// TwinCAT 3 PLC project Units
// ProgramVersion: 3.1.4023.0
// libraries:
//   tc-tools, * (hganchev)
//   Tc2_Standard, * (Beckhoff Automation GmbH)
//   Tc2_System, * (Beckhoff Automation GmbH)
//   Tc3_Module, * (Beckhoff Automation GmbH)
//   TcUnit, * (www.tcunit.org)
// project tree:
//   / PlcTask.TcTTO
//   POUs/ UnitTests.TcPOU
//   Units/ FB_TestRange.TcPOU, FB_TestRound.TcPOU, FB_TestSplit.TcPOU
// real-time tasks:
//   TASK PlcTask: cycle T#10ms, priority 20, ADS port 350

CONFIGURATION Units
    RESOURCE PLC ON TwinCAT3
        TASK PlcTask(INTERVAL := T#10ms, PRIORITY := 20);
        PROGRAM UnitTests WITH PlcTask : UnitTests;
    END_RESOURCE
END_CONFIGURATION

// ---- POUs/UnitTests.TcPOU
PROGRAM UnitTests
VAR
	fbTestRound		: Fb_TestRound;
	fbTestSplit		: FB_TestSplit;
	fbTestRange		: FB_TestRange;
END_VAR

TcUnit.RUN();

END_PROGRAM

// ---- Units/FB_TestRound.TcPOU
FUNCTION_BLOCK FB_TestRound EXTENDS TcUnit.FB_TestSuite

//REAL
testRoundRealFail();
testRoundRealSuccess();
testRoundRealToHigh();
testRoundRealToHigh2();

// LREAL
testRoundLREALFail();
testRoundLREALSuccess();
testRoundLREALToHigh();
testRoundLREALToHigh2();

METHOD testRoundLREALFail
VAR
	rValue 		: LREAL := 1000.222222;
	Actual		: LREAL;
	Expected  	: LREAL;
END_VAR
TEST('testRoundLREALFail');

// Act
Actual := 1000.222; 

// Arrange
Expected := 1000.22;

// Assert
AssertFalse( Condition := Expected = Actual, 
			 Message := 'testRoundLREALFail Failed to round LREAL');
			 
			 
			 
TEST_FINISHED();
END_METHOD

METHOD testRoundLREALSuccess
VAR
	rValue 		: LREAL := 1000.222222;
	Actual		: LREAL;
	Expected  	: LREAL;
END_VAR
TEST('testRoundLREALSuccess');

// Act
Actual := F_ROUND_LREAL(rValue, 2); 

// Arrange
Expected := 1000.22;

// Assert
AssertEquals(Expected := Expected, 
			 Actual := Actual,
			 Message := 'testRoundLREALSuccess Failed to round LREAL');
			 
			 
			 
TEST_FINISHED();
END_METHOD

METHOD testRoundLREALToHigh
VAR
	rValue 		: LREAL := 1000.226666;
	Actual		: LREAL;
	Expected  	: LREAL;
END_VAR
TEST('testRoundLREALToHigh');

// Act
Actual := F_ROUND_LREAL(rValue, 2); 

// Arrange
Expected := 1000.23;

// Assert
AssertEquals_LREAL( Expected :=  Expected, 
				Actual := Actual,
				Delta := 0.00,
			 	Message := 'testRoundLREALToHigh Failed to round LREAL');
			 
			 
			 
TEST_FINISHED();
END_METHOD

METHOD testRoundLREALToHigh2
VAR
	rValue 		: LREAL := 1000.95;
	Actual		: LREAL;
	Expected  	: LREAL;
END_VAR
TEST('testRoundLREALToHigh2');

// Act
Actual := F_ROUND_LREAL(rValue, 1); 

// Arrange
Expected := 1001.0;

// Assert
AssertEquals_LREAL( Expected :=  Expected, 
				Actual := Actual,
				Delta := 0.00,
			 	Message := 'testRoundLREALToHigh2 Failed to round LREAL');
			 
			 
			 
TEST_FINISHED();
END_METHOD

METHOD testRoundRealFail
VAR
	rValue 		: REAL := 1000.222222;
	Actual		: REAL;
	Expected  	: REAL;
END_VAR
TEST('testRoundRealFail');

// Act
Actual := 1000.222; 

// Arrange
Expected := 1000.22;

// Assert
AssertFalse( Condition := Expected = Actual, 
			 Message := 'testRoundRealFail Failed to round REAL');
			 
			 
			 
TEST_FINISHED();
END_METHOD

METHOD testRoundRealSuccess
VAR
	rValue 		: REAL := 1000.22222;
	Actual		: REAL;
	Expected  	: REAL;
END_VAR
TEST('testRoundRealSuccess');

// Act
Actual := F_ROUND_REAL(rValue, 2); 

// Arrange
Expected := 1000.22;

// Assert
AssertEquals(Expected := Expected, 
			 Actual := Actual,
			 Message := 'testRoundRealSuccess Failed to round REAL');
			 
			 
			 
TEST_FINISHED();
END_METHOD

METHOD testRoundRealToHigh
VAR
	rValue 		: REAL := 1000.226666;
	Actual		: REAL;
	Expected  	: REAL;
END_VAR
TEST('testRoundRealToHigh');

// Act
Actual := F_ROUND_REAL(rValue, 2); 

// Arrange
Expected := 1000.23;

// Assert
AssertEquals_REAL( Expected :=  Expected, 
				Actual := Actual,
				Delta := 0.00,
			 	Message := 'testRoundRealToHigh Failed to round REAL');
			 
			 
			 
TEST_FINISHED();
END_METHOD

METHOD testRoundRealToHigh2
VAR
	rValue 		: REAL := 1000.95;
	Actual		: REAL;
	Expected  	: REAL;
END_VAR
TEST('testRoundRealToHigh2');

// Act
Actual := F_ROUND_REAL(rValue, 1); 

// Arrange
Expected := 1001.0;

// Assert
AssertEquals_REAL( Expected :=  Expected, 
				Actual := Actual,
				Delta := 0.00,
			 	Message := 'testRoundRealToHigh2 Failed to round REAL');
			 
			 
			 
TEST_FINISHED();
END_METHOD

END_FUNCTION_BLOCK

// ---- Units/FB_TestSplit.TcPOU
FUNCTION_BLOCK FB_TestSplit EXTENDS TcUnit.FB_TestSuite

testSplit();

METHOD testSplit : BOOL
VAR
	sToSplit		: STRING(255) := 'Hello,this,is,split,test';
	sSplit			: ARRAY[0..Parameters.iSplitArraySize] OF STRING(255);
	sExpected		: ARRAY[0..Parameters.iSplitArraySize] OF STRING(255) := ['Hello', 'this', 'is', 'split', 'test'] ;
	
	i				: INT;
END_VAR
Test('testSplit');
// Arrange

// Act
sSplit := F_STRING_SPLIT(sToSplit, ',');

// Assert
FOR i := 0 TO Parameters.iSplitArraySize DO
	AssertEquals_STRING( Expected := sExpected[i],
				  Actual := sSplit[i],
				  Message := CONCAT('testSplit Failed to split : ', sToSplit));
END_FOR
			 
			 
TEST_FINISHED();
END_METHOD

END_FUNCTION_BLOCK

// ---- Units/FB_TestRange.TcPOU
FUNCTION_BLOCK FB_TestRange EXTENDS TcUnit.FB_TestSuite

testRange100to1000_min();
testRange100to1000_max();
testRange100to1000_mid();

METHOD testRange100to1000_max
VAR
	iValue		: INT := 100;
	
	iValue_Max	: INT := 100;
	iValue_min	: INT := 0;
	
	iRange_max	: INT := 1000;
	iRange_min	: INT := 100;
	
	Actual		: INT;
	Expected  	: INT;
	
	ActualVarInfo : __SYSTEM.VAR_INFO;
END_VAR
TEST('testRange100to1000_max');

// Act
Actual := F_GET_INT_IN_RANGE(iValue, iRange_Max, iRange_Min, iValue_Max, iValue_Min); 

// Arrange
Expected := 1000;

// Assert
AssertEquals_INT( Expected := Expected, 
				  Actual := Actual,
			 	  Message := 'testRange100to1000_max Failed to get in range INT');

ActualVarInfo :=__VARINFO(Actual);
 
AssertTrue(  Condition := ActualVarInfo.TypeName = 'INT',
			  Message := 'testRange100to1000_max Failed in type INT');
			 
			 
			 
TEST_FINISHED();
END_METHOD

METHOD testRange100to1000_mid
VAR
	iValue		: INT := 50;
	
	iValue_Max	: INT := 100;
	iValue_min	: INT := 0;
	
	iRange_max	: INT := 1000;
	iRange_min	: INT := 100;
	
	Actual		: INT;
	Expected  	: INT;
END_VAR
TEST('testRange100to1000_mid');

// Act
Actual := F_GET_INT_IN_RANGE(iValue, iRange_Max, iRange_Min, iValue_Max, iValue_Min); 

// Arrange
Expected := 550;

// Assert
AssertEquals_INT( Expected := Expected, 
				  Actual := Actual,
			 	  Message := 'testRange100to1000_mid Failed to get in range INT');
			 
			 
			 
TEST_FINISHED();
END_METHOD

METHOD testRange100to1000_min
VAR
	iValue		: INT := 0;
	
	iValue_Max	: INT := 100;
	iValue_min	: INT := 0;
	
	iRange_max	: INT := 1000;
	iRange_min	: INT := 100;
	
	Actual		: INT;
	Expected  	: INT;
END_VAR
TEST('testRange100to1000_min');

// Act
Actual := F_GET_INT_IN_RANGE(iValue, iRange_Max, iRange_Min, iValue_Max, iValue_Min); 

// Arrange
Expected := 100;

// Assert
AssertEquals_INT( Expected := Expected, 
				  Actual := Actual,
			 	  Message := 'testRange100to1000_min Failed to get in range INT');
			 
			 
			 
TEST_FINISHED();
END_METHOD

END_FUNCTION_BLOCK
